(* IEC 61131-3 sources: CodesysTest/export/Motion/Base/Axis_REF.pou/DriveEnabled.prop, 1 file *)

(* ---- Get.pm.st ---- *)
(*#-#-#-#-#-#-#-#-#-#---Declaration---#-#-#-#-#-#-#-#-#-#-#-#-#*)

VAR
END_VAR
(*#-#-#-#-#-#-#-#-#-#---Implementation---#-#-#-#-#-#-#-#-#-#-#-#-#*)

DriveEnabled := DriveEnable;
